TYPE ST_TempMeasure :
STRUCT
END_STRUCT
END_TYPE

(* stored: Version 1.1.0.1, ProductVersion 3.1.4024.12
   DUT ST_TempMeasure: Id {7116fa28-89d3-4583-a785-78a24c5a766c} *)
